// SIMATIC S7-200 project (STEP 7-Micro/WIN), CPU 221 REL 01.10

ORGANIZATION_BLOCK 主程序:OB1
TITLE=5台电动机设计的顺序启动控制系统实例
// 当操作员按下启动按钮时，电动机1控制信号立即激活，第一台电动机启动，同时触发启动间隔定时器开始计时，预设值为300。启动间隔定时器仅在电动机5控制信号未激活时开始计时，确保启动过程按顺序进行。
// 当启动间隔定时器计时到50时，电动机2控制信号必须激活，启动第二台电动机；计时到100时，电动机3控制信号必须激活，启动第三台电动机；计时到150时，电动机4控制信号必须激活，启动第四台电动机；计时到200时，电动机5控制信号必须激活，启动第五台电动机。整个启动过程在20秒内完成，从电动机1控制信号到电动机5控制信号逐一激活。
// 所有电动机启动后，启动间隔定时器仍继续计时至300。
// 若操作员按下停止按钮，电动机1、2、3、4、5控制信号必须立即复位。
// 顺序启动过程在20秒内完成，从第一台电动机到第五台电动机逐一激活。
// 若启动按钮保持接通，电动机1控制信号必须持续激活，直到停止按钮触发。
BEGIN
Network 1 // 网络标题
// 网络注释：按下启动按钮第一台电动机启动。
LD     I0.0
O      Q0.0
=      Q0.0
AN     Q0.4
TON    T37, 300
Network 2
// 网络注释：5S时,第二台电动机启动
LDW>=  T37, 50
S      Q0.1, 1
Network 3
// 网络注释;10S时,第三台电动机启动
LDW>=  T37, 100
S      Q0.2, 1
Network 4
// 网络注释：15S时，第4台电动机启动
LDW>=  T37, 150
S      Q0.3, 1
Network 5
// 网络注释：20S时，第5台电动机启动
LDW>=  T37, 200
S      Q0.4, 1
Network 6
// 网络注释：按下停止按钮，5台电动机停止
LDN    I0.1
R      Q0.0, 5
END_ORGANIZATION_BLOCK
